(* IEC 61131-3 sources: ae-tiax/src/Trafficlight, 7 files *)

(* ---- Colors.st ---- *)
NAMESPACE Simatic.Ax.Tiax
    TYPE
        Colors : (RED, GREEN, YELLOW, RED_YELLOW) := RED;
    END_TYPE
END_NAMESPACE

(* ---- AbstractTrafficLightState.st ---- *)
USING Simatic.Ax.StateFramework;

NAMESPACE Simatic.Ax.Tiax

    // Abstract class
    CLASS ABSTRACT AbstractTrafficLightState
        EXTENDS State1Transition // class from external AX package @simatic-ax/statemachine

        // private static
        VAR
            count : LINT;
            activations : LINT;
        END_VAR

        /// Public method to return the number of activations
        METHOD PUBLIC GetActivations : LINT;
            GetActivations := activations;
        END_METHOD

        /// Public method to return the number of calls
        METHOD PUBLIC GetCalls : LINT;
            GetCalls := count;
        END_METHOD

        /// public abstract method with return value which has to be implemented inthe concrete class
        METHOD PUBLIC ABSTRACT GetColor : Colors
        END_METHOD
    END_CLASS

END_NAMESPACE

(* ---- StateGreen.st ---- *)
USING Simatic.Ax.StateFramework;

NAMESPACE Simatic.Ax.Tiax

    CLASS StateGreen
        EXTENDS AbstractTrafficLightState // inherit from AbstractTrafficLightState

        // public static
        VAR PUBLIC
            gn : REF_TO BOOL; //Reference
        END_VAR

        // public method with non return value
        METHOD PUBLIC OVERRIDE OnEntry
            activations := activations + 1;
            gn^ := TRUE; // dereference
        END_METHOD

        // public method with non return value
        METHOD PUBLIC OVERRIDE Action
            count := count + 1;
        END_METHOD

        // public method with non return value
        METHOD PUBLIC OVERRIDE OnExit
            gn^ := FALSE; // dereference
        END_METHOD

        // public method with return value
        METHOD PUBLIC OVERRIDE GetColor : Colors
            GetColor := Colors#Green; // set return value to enum value green
        END_METHOD
    END_CLASS

END_NAMESPACE

(* ---- StateRed.st ---- *)
USING Simatic.Ax.StateFramework;

NAMESPACE Simatic.Ax.Tiax

    CLASS StateRed
        EXTENDS State1Transition
        VAR
            count : LINT;
            activations : LINT;
        END_VAR
        VAR PUBLIC
            rd : REF_TO BOOL;
        END_VAR
        METHOD PUBLIC OVERRIDE OnEntry
            activations := activations + 1;
            rd^ := TRUE;
        END_METHOD
        METHOD PUBLIC OVERRIDE Action
            count := count + 1;
        END_METHOD
        METHOD PUBLIC OVERRIDE OnExit
            rd^ := FALSE;
        END_METHOD
        METHOD PUBLIC GetColor : Colors
            GetColor := Colors#Red;
        END_METHOD
    END_CLASS

END_NAMESPACE

(* ---- StateRedYellow.st ---- *)
USING Simatic.Ax.StateFramework;

NAMESPACE Simatic.Ax.Tiax

    CLASS StateRedYellow
        EXTENDS AbstractTrafficLightState // inherit from AbstractTrafficLightState
        VAR PUBLIC
            rd : REF_TO BOOL;
            ye : REF_TO BOOL;
        END_VAR
        METHOD PUBLIC OVERRIDE OnEntry
            activations := activations + 1;
            rd^ := TRUE;
            ye^ := TRUE;
        END_METHOD
        METHOD PUBLIC OVERRIDE Action
            count := count + 1;
        END_METHOD
        METHOD PUBLIC OVERRIDE OnExit
            rd^ := FALSE;
            ye^ := FALSE;
        END_METHOD
        METHOD PUBLIC OVERRIDE GetColor : Colors
            GetColor := Colors#Red_Yellow;
        END_METHOD
    END_CLASS

END_NAMESPACE

(* ---- StateYellow.st ---- *)
USING Simatic.Ax.StateFramework;

NAMESPACE Simatic.Ax.Tiax

    CLASS StateYellow
        EXTENDS State1Transition
        VAR PUBLIC
            ye : REF_TO BOOL;
        END_VAR
        VAR
            count : LINT;
            activations : LINT;
        END_VAR
        METHOD PUBLIC OVERRIDE OnEntry
            activations := activations + 1;
            ye^ := TRUE;
        END_METHOD
        METHOD PUBLIC OVERRIDE Action
            count := count + 1;
        END_METHOD
        METHOD PUBLIC OVERRIDE OnExit
            ye^ := FALSE;
        END_METHOD
        METHOD PUBLIC GetColor : Colors
            GetColor := Colors#Yellow;
        END_METHOD
    END_CLASS

END_NAMESPACE

(* ---- TrafficlightWrapper.st ---- *)
USING Simatic.Ax.StateFramework;

NAMESPACE Simatic.Ax.Tiax
    // Wrapper for TIA Portal usage
    FUNCTION_BLOCK TrafficlightWrapper
        VAR_OUTPUT
            activeStateId : INT;
            status : StateControllerStatus;
            rd : BOOL;
            ye : BOOL;
            gn : BOOL;
        END_VAR
        VAR
            _sc : StateController;
            _stateRed : StateRed;
            _stateRedTrans : Transition;
            _TimeoutGuard : TimeoutGuard;
            _stateRedYellow : StateRedYellow;
            _stateRedYellowTrans : Transition;
            _stateGreen : StateGreen;
            _stateGreenTrans : Transition;
            _stateYellow : StateYellow;
            _stateYellowTrans : Transition;
            init : BOOL;
        END_VAR

        IF NOT init THEN
            // Congfigure StateController
            _sc.InitialState := _stateRed;
            _TimeoutGuard.Timeout := T#1000ms;
            // Configure Red
            _stateRed.Transition1 := _stateRedTrans;
            _stateRed.StateID := 1;
            _stateRedTrans.NextState := _stateRedYellow;
            _stateRedTrans.Guard := _TimeoutGuard;
            _stateRed.rd := REF(rd);
            // Configure RedYellow
            _stateRedYellow.Transition1 := _stateRedYellowTrans;
            _stateRedYellow.StateID := 2;
            _stateRedYellowTrans.NextState := _stateGreen;
            _stateRedYellowTrans.Guard := _TimeoutGuard;
            _stateRedYellow.rd := REF(rd);
            _stateRedYellow.ye := REF(ye);
            // Configure Green
            _stateGreen.Transition1 := _stateGreenTrans;
            _stateGreen.StateID := 3;
            _stateGreenTrans.NextState := _stateYellow;
            _stateGreenTrans.Guard := _TimeoutGuard;
            _stateGreen.gn := REF(gn);
            // Configure Yellow
            _stateYellow.Transition1 := _stateYellowTrans;
            _stateYellow.StateID := 4;
            _stateYellowTrans.NextState := _stateRed;
            _stateYellowTrans.Guard := _TimeoutGuard;
            _stateYellow.ye := REF(ye);
            init := TRUE;
        END_IF;
        _sc.Execute();
        status := _sc.GetState();
    END_FUNCTION_BLOCK

END_NAMESPACE
